TYPE T_TriggerControl :
UNION
  Ctrl         : BYTE;
  Bits         : T_TriggerControlBits;
END_UNION
END_TYPE

(* stored: Version 1.1.0.1, ProductVersion 3.1.4024.12
   DUT T_TriggerControl: Id {fc584296-b9a7-49d5-be97-39d776e36b2b} *)
